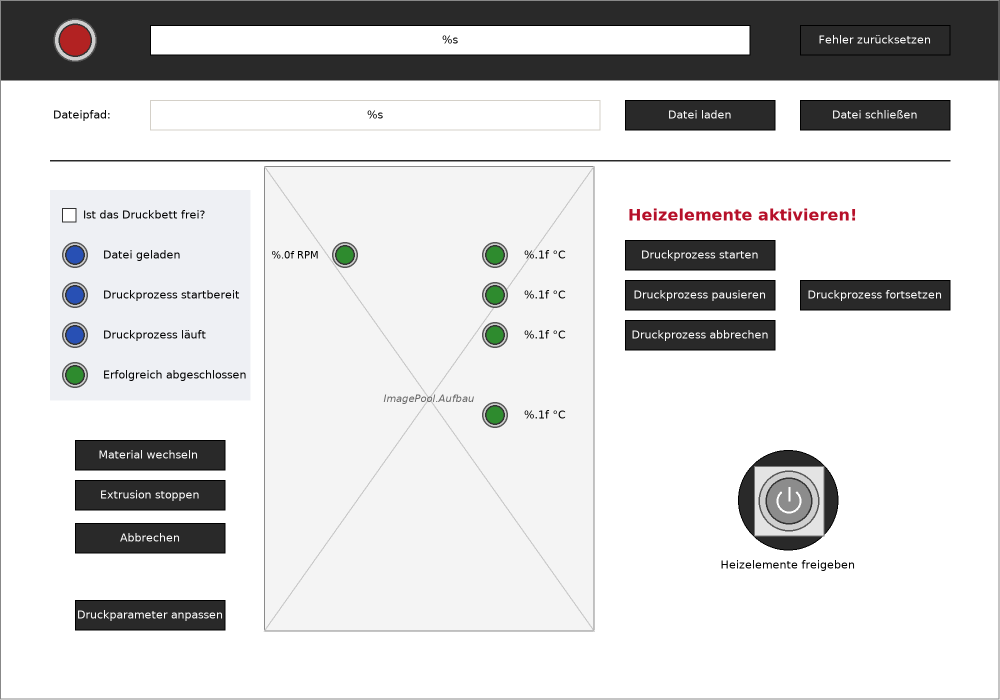
VISUALIZATION V_Homescreen  // 1000x700
    Rectangle (625,100 150x30), "Datei laden", colour toggle: GVL_ProgramSequencer.Sequencer.bLoadFile, input disabled if: Sequencer.bFileLoaded
        OnMouseDown: toggle GVL_ProgramSequencer.Sequencer.bLoadFile
    Textfield (150,100 450x30), "%s", text variable: GVL_ProgramSequencer.Sequencer.sPath
        OnMouseDown: write the text variable via Default, format %s
    Label (50,100 100x30), "Dateipfad:"
    Rectangle (800,100 150x30), "Datei schließen", colour toggle: GVL_ProgramSequencer.Sequencer.bCloseFile, input disabled if: NOT Sequencer.bFileLoaded OR GVL_ProgramSequencer.Sequencer.bPrinting
        OnMouseDown: toggle GVL_ProgramSequencer.Sequencer.bCloseFile
    Group (713,450 150x130)
        Ellipse (25,0 100x100), colour toggle: GVL_ProgramSequencer.Sequencer.bHeatersEnabled
        PowerSwitch (41,16 70x70), variable: GVL_ProgramSequencer.Sequencer.bHeatersEnabled, behaviour: TOGGLE, style: Switch-PowerSwitch-Gray
        Label (0,100 150x30), "Heizelemente freigeben"
    Rectangle (625,240 150x30), "Druckprozess starten", colour toggle: GVL_ProgramSequencer.Sequencer.bStart, invisible if: Sequencer.eState < E_StateSequencer.READY OR Sequencer.eState >= E_StateSequencer.SHUTDOWN, input disabled if: Sequencer.eState > E_StateSequencer.READY
        OnMouseDown: toggle GVL_ProgramSequencer.Sequencer.bStart
    Label (625,200 262x30), "Heizelemente aktivieren!", invisible if: GVL_ProgramSequencer.Sequencer.bHeatersEnabled OR (Sequencer.eState < E_StateSequencer.IDLE OR Sequencer.eState >= E_StateSequencer.SHUTDOWN)
    Rectangle (625,280 150x30), "Druckprozess pausieren", colour toggle: GVL_ProgramSequencer.Sequencer.bPause, invisible if: Sequencer.eState < E_StateSequencer.READY OR Sequencer.eState >= E_StateSequencer.SHUTDOWN, input disabled if: Sequencer.eState = E_StateSequencer.PAUSE
        OnMouseDown: toggle GVL_ProgramSequencer.Sequencer.bPause
    Rectangle (800,280 150x30), "Druckprozess fortsetzen", colour toggle: GVL_ProgramSequencer.Sequencer.bResume, invisible if: Sequencer.eState < E_StateSequencer.READY OR Sequencer.eState >= E_StateSequencer.SHUTDOWN, input disabled if: Sequencer.eState <> E_StateSequencer.PAUSE
        OnMouseDown: toggle GVL_ProgramSequencer.Sequencer.bResume
    Rectangle (625,320 150x30), "Druckprozess abbrechen", invisible if: Sequencer.eState < E_StateSequencer.READY OR Sequencer.eState >= E_StateSequencer.SHUTDOWN, input disabled if: GVL_ProgramSequencer.Sequencer.bAbort
        OnMouseDown: toggle GVL_ProgramSequencer.Sequencer.bAbort
    Group (0,0 1000x80)
        Rectangle (0,0 1000x80)
        Rectangle (800,25 150x30), "Fehler zurücksetzen", colour toggle: GVL_ProgramSequencer.Sequencer.bError
            OnMouseDown: execute { GVL_ProgramSequencer.Sequencer.bErrorReset := TRUE; }
        Lamp1 (50,15 50x50), variable: GVL_ProgramSequencer.Sequencer.bError, style: Lamp-Lamp1-Red
        Rectangle (150,25 600x30), "%s", text variable: GVL_ProgramSequencer.Sequencer.sErrorMsg
    Rectangle (50,160 900x1)
    Rectangle (75,600 150x30), "Druckparameter anpassen"
        OnMouseDown: change screen: V_Konfiguration
    Rectangle (75,440 150x30), "Material wechseln", colour toggle: GVL_ProgramSequencer.Sequencer.bResume, invisible if: Sequencer.eState >= E_StateSequencer.READY, input disabled if: Sequencer.eState <> E_StateSequencer.IDLE
        OnMouseDown: toggle GVL_ProgramSequencer.Sequencer.bChangeMaterial
    Rectangle (50,190 200x210)
    Label (100,280 140x30), "Druckprozess startbereit"
    Lamp1 (60,280 30x30), variable: GVL_ProgramSequencer.Sequencer.bPrintBedClear AND GVL_ProgramSequencer.Sequencer.bReady, style: Lamp-Lamp1-Blue
    Label (100,320 140x30), "Druckprozess läuft"
    Lamp1 (60,320 30x30), variable: GVL_ProgramSequencer.Sequencer.bPrinting, style: Lamp-Lamp1-Blue
    Label (100,360 140x30), "Erfolgreich abgeschlossen"
    Lamp1 (60,360 30x30), variable: GVL_ProgramSequencer.Sequencer.bFinished, style: Lamp-Lamp1-Green
    Label (100,240 140x30), "Datei geladen"
    Lamp1 (60,240 30x30), variable: Sequencer.bFileLoaded, style: Lamp-Lamp1-Blue
    Checkbox (60,200 185x30), "Ist das Druckbett frei?", variable: GVL_ProgramSequencer.Sequencer.bPrintBedClear
    Rectangle (75,480 150x30), "Extrusion stoppen", colour toggle: GVL_ProgramSequencer.Sequencer.bResume, invisible if: Sequencer.eState >= E_StateSequencer.READY, input disabled if: Sequencer.eState <> E_StateSequencer.CHANGE_MATERIAL_2
        OnMouseDown: toggle GVL_ProgramSequencer.Sequencer.bChangeMaterialFinished
    Image (264,166 330x465), image: ImagePool.Aufbau
    Lamp1 (330,240 30x30), variable: GVL_Extruder.Extruder.bExtruding, style: Lamp-Lamp1-Green
    Rectangle (75,523 150x30), "Abbrechen", invisible if: Sequencer.eState >= E_StateSequencer.READY, input disabled if: Sequencer.eState <= E_StateSequencer.IDLE
        OnMouseDown: toggle GVL_ProgramSequencer.Sequencer.bAbort
    Rectangle (520,240 50x30), "%.1f °C", text variable: GVL_Extruder.HeaterTop.fActualTemp
    Rectangle (520,280 50x30), "%.1f °C", text variable: GVL_Extruder.HeaterMiddle.fActualTemp
    Rectangle (520,320 50x30), "%.1f °C", text variable: GVL_Extruder.HeaterNozzle.fActualTemp
    Lamp1 (480,240 30x30), variable: GVL_Extruder.HeaterTop.bAtTemp, style: Lamp-Lamp1-Green
    Lamp1 (480,280 30x30), variable: GVL_Extruder.HeaterMiddle.bAtTemp, style: Lamp-Lamp1-Green
    Lamp1 (480,320 30x30), variable: GVL_Extruder.HeaterNozzle.bAtTemp, style: Lamp-Lamp1-Green
    Rectangle (270,240 50x30), "%.0f RPM", text variable: ExtruderMotor.fDisplay_RPM
    Rectangle (520,400 50x30), "%.1f °C", text variable: GVL_PrintingBed.PrintingBed.fActualTemp
    Lamp1 (480,400 30x30), variable: GVL_PrintingBed.PrintingBed.bAtTemp, style: Lamp-Lamp1-Green
END_VISUALIZATION

(* stored: Version 1.1.0.1
   Visu V_Homescreen: Id {ba2c5013-d3ca-45a8-ba17-2f925d7fdcb5} *)
